FUNCTION_BLOCK FB_SlitPair_ISIS
VAR_INPUT
    nIdPositiveAxis: UINT; //ID of axis for which positive motion increases gap size
    nIdNegativeAxis: UINT; //ID of axis for which negative motion increases gap size
    nIdGapSizeAxis: UINT; //ID of virtual gap aperture size axis
    nIdGapCentreAxis: UINT; //ID of virtual gap centre position axis

    bEnable: BOOL; //Enable slit pair logic functionality
    bReset: BOOL; //Reset from error state
    fEncoderScaling: LREAL := 10000; //Virtual axis scaling denominator, default of 10000
    
    
    
END_VAR

//Linkable objects
VAR
    //Replacement limit links for real axes
    bPositiveAxis_FwdLimit AT %I* : BOOL;
    bPositiveAxis_BwdLimit AT %I* : BOOL;
    bNegativeAxis_FwdLimit AT %I* : BOOL;
    bNegativeAxis_BwdLimit AT %I* : BOOL;
    
    //Software encoders for virtual axes
    nGapSizeEncoder AT %Q*: UDINT := 0;
    nGapCentreEncoder AT %Q*: UDINT := 0;
END_VAR

VAR   
    fGapSize: LREAL;
    fGapCentre: LREAL;
    
    bAllHalted: BOOL := FALSE;
    bInternalResetHome: BOOL :=FALSE;

    fbSetpointGenEnablePositiveAxis: MC_ExtSetPointGenEnable;
    fbSetpointGenEnableNegativeAxis: MC_ExtSetPointGenEnable;
    fbSetpointGenEnableGapSizeAxis: MC_ExtSetPointGenEnable;
    fbSetpointGenEnableGapCentreAxis: MC_ExtSetPointGenEnable;

    fbSetpointGenDisablePositiveAxis: MC_ExtSetPointGenDisable;
    fbSetpointGenDisableNegativeAxis: MC_ExtSetPointGenDisable;
    fbSetpointGenDisableGapSizeAxis: MC_ExtSetPointGenDisable;
    fbSetpointGenDisableGapCentreAxis: MC_ExtSetPointGenDisable;

    fPosSetpointPositiveAxis: LREAL;
    fPosSetpointNegativeAxis: LREAL;
    fPosSetpointGapSizeAxis: LREAL;
    fPosSetpointGapCentreAxis: LREAL;
    
    fPosSetpointPositiveAxis_Nominal: LREAL;
    fPosSetpointNegativeAxis_Nominal: LREAL;
    fPosSetpointGapSizeAxis_Nominal: LREAL;
    fPosSetpointGapCentreAxis_Nominal: LREAL;

    fVeloSetpointPositiveAxis: LREAL;
    fVeloSetpointNegativeAxis: LREAL;
    fVeloSetpointGapSizeAxis: LREAL;
    fVeloSetpointGapCentreAxis: LREAL;

    fVeloSetpointPositiveAxis_Nominal: LREAL;
    fVeloSetpointNegativeAxis_Nominal: LREAL;
    fVeloSetpointGapSizeAxis_Nominal: LREAL;
    fVeloSetpointGapCentreAxis_Nominal: LREAL;
    
    nDirectionPositiveAxis: DINT;
    nDirectionNegativeAxis: DINT;
    nDirectionGapSizeAxis: DINT;
    nDirectionGapCentreAxis: DINT;
    
    ePositiveAxisState : E_AxisLimitState;
    eNegativeAxisState : E_AxisLimitState;
    eAxisPairState : E_SlitPairLimitState;
    

    eState: E_SlitPairStates := E_SlitPairStates.eInit;

    bInternalReset: BOOL;
    bHomingReset: BOOL := FALSE;

    //Two resets required due to homing functionality
    bResetInProgressCheck1: BOOL := FALSE;
    bResetInProgressCheck2: BOOL := FALSE;

    //internal MC_Reset, needed because the current reset in FB_Axis works only when there is an error. This should change once the reset functionality changes
    fbInternalResetTrig: R_TRIG;
    fbInternalResetHome: R_TRIG;
    fbResetPositiveAxis: MC_RESET;
    fbResetNegativeAxis: MC_RESET;
    fbResetGapSizeAxis: MC_RESET;
    fbResetGapCentreAxis: MC_RESET;
    fbResetHomedGap: MC_Home;
    fbResetHomedCentre: MC_Home;

END_VAR

(*SETUP INSTRUCTIONS
    All Axes:
        Allow motion commands to external setpoint axis := FALSE;
    Real Axes:
        Do not link limit switches to astAxes struct. Limits must be linked to FB_SlitPair_ISIS inputs
    Virtual axes:
        Encoder type set to Encoder (universal)
        Encoder mask set to 0xFFFFFFFF
        Encoder numerator/denominator scaling set to match FB fEncoderScaling value (default of 10 000 results in numerator of 0.0001 with denominator of 1)
        Link nDataIn1 of encoder to FB encoders
        Position lag monitoring can be left on
        Dynamics of virtual axes must be configured considering coupled mechanicals (e.g. don't set velocities your real axes can't achieve)
*)

//Limit switch passthrough by default - overridden where required in later logic to satisfy ExternalSetpointGenerators
GVL.astAxes[nIdPositiveAxis].stInputs.bLimitFwd:= bPositiveAxis_FwdLimit;
GVL.astAxes[nIdPositiveAxis].stInputs.bLimitBwd:= bPositiveAxis_BwdLimit;
GVL.astAxes[nIdNegativeAxis].stInputs.bLimitFwd:= bNegativeAxis_FwdLimit;
GVL.astAxes[nIdNegativeAxis].stInputs.bLimitBwd:= bNegativeAxis_BwdLimit;

//Enable Logic - Virtual axes automatically enable when real axes are enabled
actVirtualAxisEnable();

//Position of virtual axes
actVirtualAxisPositions();

//Determine limit state of real axes
actLimitState();

//Set fwEnabled and bwEnabled of virtual axes
actVirtualAxisLimits();

//Calculate position and velocity setpoints
actCalculateSetpointPositionAndVelocity();

//Calculate direction setpoints
actCalculateSetpointDirections();




//Error state handling - only handle errors that disable motion
IF bEnable AND (GVL.astAxes[nIdPositiveAxis].Axis.Status.ErrorStop OR GVL.astAxes[nIdNegativeAxis].Axis.Status.ErrorStop OR GVL.astAxes[nIdGapSizeAxis].Axis.Status.ErrorStop OR GVL.astAxes[nIdGapCentreAxis].Axis.Status.ErrorStop) THEN
    eState := E_SlitPairStates.eError;
END_IF

//Propagate real axis error to virtual
IF GVL.astAxes[nIdPositiveAxis].Axis.Status.ErrorStop AND (NOT GVL.astAxes[nIdGapSizeAxis].Axis.Status.ErrorStop OR NOT GVL.astAxes[nIdGapCentreAxis].Axis.Status.ErrorStop) THEN
    GVL.astAxes[nIdGapSizeAxis].stStatus.bError := TRUE;
    GVL.astAxes[nIdGapCentreAxis].stStatus.bError := TRUE;
    GVL.astAxes[nIdGapSizeAxis].stStatus.nErrorID := GVL.astAxes[nIdPositiveAxis].stStatus.nErrorID;
    GVL.astAxes[nIdGapCentreAxis].stStatus.nErrorID := GVL.astAxes[nIdPositiveAxis].stStatus.nErrorID;
ELSIF  GVL.astAxes[nIdNegativeAxis].Axis.Status.ErrorStop AND (NOT GVL.astAxes[nIdGapSizeAxis].Axis.Status.ErrorStop OR NOT GVL.astAxes[nIdGapCentreAxis].Axis.Status.ErrorStop) THEN
    GVL.astAxes[nIdGapSizeAxis].stStatus.bError := TRUE;
    GVL.astAxes[nIdGapCentreAxis].stStatus.bError := TRUE;
    GVL.astAxes[nIdGapSizeAxis].stStatus.nErrorID := GVL.astAxes[nIdNegativeAxis].stStatus.nErrorID;
    GVL.astAxes[nIdGapCentreAxis].stStatus.nErrorID := GVL.astAxes[nIdNegativeAxis].stStatus.nErrorID;
END_IF

//Internal Reset linked to any axis reset
bInternalReset := bReset OR GVL.astAxes[nIdPositiveAxis].stControl.bReset OR GVL.astAxes[nIdNegativeAxis].stControl.bReset OR GVL.astAxes[nIdGapSizeAxis].stControl.bReset OR GVL.astAxes[nIdGapCentreAxis].stControl.bReset;

//If real axis is homing, change state
IF bEnable AND (GVL.astAxes[nIdPositiveAxis].Axis.Status.HomingBusy OR GVL.astAxes[nIdNegativeAxis].Axis.Status.HomingBusy) THEN
    eState := E_SlitPairStates.eWaitForRealHomed;
END_IF

//Link all halt buttons in motors
IF GVL.astAxes[nIdPositiveAxis].stControl.bHalt OR GVL.astAxes[nIdNegativeAxis].stControl.bHalt OR
    GVL.astAxes[nIdGapSizeAxis].stControl.bHalt OR GVL.astAxes[nIdGapCentreAxis].stControl.bHalt THEN
    actHaltAllAxes();   //Will upset setpoint generator axes - may be able to fix by only issuing to non-setpoint generated axes
END_IF

//Propagate homing status
fbResetHomedGap(Axis:= GVL.astAxes[nIdGapSizeAxis].Axis, HomingMode:= MC_ResetCalibration);
fbResetHomedCentre(Axis:= GVL.astAxes[nIdGapCentreAxis].Axis, HomingMode:= MC_ResetCalibration);
fbInternalResetHome(CLK:= fbResetHomedCentre.Done OR fbResetHomedGap.Done );

IF NOT GVL.astAxes[nIdPositiveAxis].stStatus.bHomed OR NOT GVL.astAxes[nIdNegativeAxis].stStatus.bHomed THEN
        fbResetHomedGap.Execute := TRUE;
        fbResetHomedCentre.Execute := TRUE;
END_IF

IF fbInternalResetHome.Q THEN
        fbResetHomedGap.Execute := FALSE;
        fbResetHomedCentre.Execute := FALSE;
END_IF


//State machine
IF bEnable THEN
    CASE eState OF  //HOMING LOOP ISSUE
        E_SlitPairStates.eInit:
            //If real axes are calibrated, then home the virtual axes, else go Operatioanl
            fbResetPositiveAxis(Axis:=GVL.astAxes[nIdPositiveAxis].Axis, Execute:=FALSE);
            fbResetNegativeAxis(Axis:=GVL.astAxes[nIdNegativeAxis].Axis, Execute:=FALSE);
            fbResetGapSizeAxis(Axis:=GVL.astAxes[nIdGapSizeAxis].Axis, Execute:=FALSE);
            fbResetGapCentreAxis(Axis:=GVL.astAxes[nIdGapCentreAxis].Axis, Execute:=FALSE);
            IF GVL.astAxes[nIdPositiveAxis].stStatus.bHomed AND GVL.astAxes[nIdNegativeAxis].stStatus.bHomed THEN
               GVL.astAxes[nIdGapSizeAxis].stConfig.eHomeSeq := E_HomingRoutines.eHomeDirect;
               GVL.astAxes[nIdGapCentreAxis].stConfig.eHomeSeq := E_HomingRoutines.eHomeDirect;
               GVL.astAxes[nIdGapSizeAxis].stConfig.fHomePosition := fGapSize;
               GVL.astAxes[nIdGapCentreAxis].stConfig.fHomePosition := fGapCentre;
                eState := E_SlitPairStates.eWaitForVirtualHomed;
            ELSE
                eState := E_SlitPairStates.eOperational;
            END_IF

        E_SlitPairStates.eWaitForVirtualHomed:
            //Wait for virtual axis homing to complete/
            GVL.astAxes[nIdGapSizeAxis].stControl.eCommand := E_MotionFunctions.eHome;
            GVL.astAxes[nIdGapSizeAxis].stControl.bExecute := TRUE;
            GVL.astAxes[nIdGapCentreAxis].stControl.eCommand := E_MotionFunctions.eHome;
            GVL.astAxes[nIdGapCentreAxis].stControl.bExecute := TRUE;
            IF GVL.astAxes[nIdGapSizeAxis].stStatus.bHomed AND GVL.astAxes[nIdGapCentreAxis].stStatus.bHomed THEN
                eState := E_SlitPairStates.eOperational;
            END_IF
            //IF NOT IN HOMING STATE

        E_SlitPairStates.eOperational:
            bResetInProgressCheck1 := FALSE;
            //Detect whether real or virtual axes are moving
            IF GVL.astAxes[nIdGapSizeAxis].stStatus.bMoving OR GVL.astAxes[nIdGapCentreAxis].stStatus.bMoving THEN
                eState := E_SlitPairStates.eEnableRealGenerators;
            END_IF
            IF GVL.astAxes[nIdPositiveAxis].stStatus.bMoving OR GVL.astAxes[nIdNegativeAxis].stStatus.bMoving THEN
                eState := E_SlitPairStates.eEnableVirtualGenerators;
            END_IF

        E_SlitPairStates.eEnableRealGenerators:
            //Temporary override of limits
            GVL.astAxes[nIdPositiveAxis].stInputs.bLimitFwd:= TRUE;
            GVL.astAxes[nIdPositiveAxis].stInputs.bLimitBwd:= TRUE;
            GVL.astAxes[nIdNegativeAxis].stInputs.bLimitFwd:= TRUE;
            GVL.astAxes[nIdNegativeAxis].stInputs.bLimitBwd:= TRUE;
            fbSetpointGenEnablePositiveAxis.Execute := TRUE;
            fbSetpointGenEnableNegativeAxis.Execute := TRUE;
            eState := E_SlitPairStates.eCheckRealAxisGeneratorsEnabled;

        E_SlitPairStates.eCheckRealAxisGeneratorsEnabled:
            //Hold MC_Power on until generators have enabled           
            IF fbSetpointGenEnablePositiveAxis.Enabled AND fbSetpointGenEnableNegativeAxis.Enabled THEN
                eState := E_SlitPairStates.eWaitForVirtualMoveDone;
            END_IF

        E_SlitPairStates.eWaitForVirtualMoveDone:            
            IF NOT(GVL.astAxes[nIdGapSizeAxis].stStatus.bMoving OR GVL.astAxes[nIdGapCentreAxis].stStatus.bMoving) THEN
                eState := E_SlitPairStates.eDisableRealGenerators;
            END_IF

        E_SlitPairStates.eDisableRealGenerators:
            fbSetpointGenDisablePositiveAxis.Execute := TRUE;
            fbSetpointGenDisableNegativeAxis.Execute := TRUE;
            eState := E_SlitPairStates.eOperational;

        E_SlitPairStates.eEnableVirtualGenerators:
            //Hold MC_Power on until generators have enabled
            GVL.astAxes[nIdPositiveAxis].stInputs.bLimitFwd:= TRUE;
            GVL.astAxes[nIdPositiveAxis].stInputs.bLimitBwd:= TRUE;
            GVL.astAxes[nIdNegativeAxis].stInputs.bLimitFwd:= TRUE;
            GVL.astAxes[nIdNegativeAxis].stInputs.bLimitBwd:= TRUE;
            fbSetpointGenEnableGapSizeAxis.Execute := TRUE;
            fbSetpointGenEnableGapCentreAxis.Execute := TRUE;
            eState := E_SlitPairStates.eCheckVirtualAxisGeneratorsEnabled;

        E_SlitPairStates.eCheckVirtualAxisGeneratorsEnabled:
            //Hold MC_Power on until generators have enabled
            IF fbSetpointGenEnableGapSizeAxis.Enabled AND fbSetpointGenEnableGapCentreAxis.Enabled THEN
                eState := E_SlitPairStates.eWaitForRealMoveDone;
            END_IF

        E_SlitPairStates.eWaitForRealMoveDone:
            IF NOT(GVL.astAxes[nIdPositiveAxis].stStatus.bMoving OR GVL.astAxes[nIdNegativeAxis].stStatus.bMoving) THEN
                eState := E_SlitPairStates.eDisableVirtualGenerators;
            END_IF

        E_SlitPairStates.eDisableVirtualGenerators:
            fbSetpointGenDisableGapSizeAxis.Execute := TRUE;
            fbSetpointGenDisableGapCentreAxis.Execute := TRUE;
            eState := E_SlitPairStates.eOperational;

        E_SlitPairStates.eError:
            actHaltAllAxes();

            IF bHomingReset THEN
                bInternalReset := TRUE;
                bResetInProgressCheck1 := TRUE;
                bResetInProgressCheck2 := TRUE;
                bHomingReset := FALSE;
            END_IF
            IF bInternalReset OR bReset OR bResetInProgressCheck2 THEN
                fbResetPositiveAxis(Axis:=GVL.astAxes[nIdPositiveAxis].Axis, Execute:=TRUE);
                fbResetNegativeAxis(Axis:=GVL.astAxes[nIdNegativeAxis].Axis, Execute:=TRUE);
                fbResetGapSizeAxis(Axis:=GVL.astAxes[nIdGapSizeAxis].Axis, Execute:=TRUE);
                fbResetGapCentreAxis(Axis:=GVL.astAxes[nIdGapCentreAxis].Axis, Execute:=TRUE);
                GVL.astAxes[nIdPositiveAxis].stControl.bReset := TRUE;
                GVL.astAxes[nIdNegativeAxis].stControl.bReset := TRUE;
                GVL.astAxes[nIdGapSizeAxis].stControl.bReset := TRUE;
                GVL.astAxes[nIdGapCentreAxis].stControl.bReset := TRUE;
                IF NOT(bResetInProgressCheck1) THEN
                    bResetInProgressCheck2 := FALSE;
                END_IF
            END_IF

            IF NOT(GVL.astAxes[nIdPositiveAxis].stStatus.bError) AND NOT(GVL.astAxes[nIdNegativeAxis].stStatus.bError) AND NOT(GVL.astAxes[nIdGapSizeAxis].stStatus.bError) AND NOT(GVL.astAxes[nIdGapCentreAxis].stStatus.bError) THEN
                eState := E_SlitPairStates.eInit;
            END_IF

        E_SlitPairStates.eWaitForRealHomed:
            bHomingReset := TRUE;
            IF NOT GVL.astAxes[nIdPositiveAxis].Axis.Status.Homed OR NOT GVL.astAxes[nIdNegativeAxis].Axis.Status.Homed THEN
                eState := E_SlitPairStates.eInit;
            END_IF
    END_CASE
END_IF

//Call spGenerator FBs
actGeneratorEnableDisable();

//Feed externalsetpoint generators setpoint values - ignoring acceleration
MC_ExtSetPointGenFeed(Axis:= GVL.astAxes[nIdPositiveAxis].Axis, Position:= fPosSetpointPositiveAxis, Velocity:= fVeloSetpointPositiveAxis, Acceleration:= 0, Direction:= nDirectionPositiveAxis);
MC_ExtSetPointGenFeed(Axis:= GVL.astAxes[nIdNegativeAxis].Axis, Position:= fPosSetpointNegativeAxis, Velocity:= fVeloSetpointNegativeAxis, Acceleration:= 0, Direction:= nDirectionNegativeAxis);
MC_ExtSetPointGenFeed(Axis:= GVL.astAxes[nIdGapSizeAxis].Axis, Position:= fPosSetpointGapSizeAxis, Velocity:= fVeloSetpointGapSizeAxis, Acceleration:= 0, Direction:= nDirectionGapSizeAxis);
MC_ExtSetPointGenFeed(Axis:= GVL.astAxes[nIdGapCentreAxis].Axis, Position:= fPosSetpointGapCentreAxis, Velocity:= fVeloSetpointGapCentreAxis, Acceleration:= 0, Direction:= nDirectionGapCentreAxis);

bReset := FALSE;

ACTION actCalculateSetpointDirections:
IF fVeloSetpointPositiveAxis > 0 THEN
    nDirectionPositiveAxis := 1; //moving forward
ELSIF fVeloSetpointPositiveAxis < 0 THEN
    nDirectionPositiveAxis := -1; //moving backward
ELSE
    nDirectionPositiveAxis := 0; //stationary
END_IF

IF fVeloSetpointNegativeAxis > 0 THEN
    nDirectionNegativeAxis := 1; //moving forward
ELSIF fVeloSetpointNegativeAxis < 0 THEN
    nDirectionNegativeAxis := -1; //moving backward
ELSE
    nDirectionNegativeAxis := 0; //stationary
END_IF

IF fVeloSetpointGapSizeAxis > 0 THEN
    nDirectionGapSizeAxis := 1; //moving forward
ELSIF fVeloSetpointGapSizeAxis < 0 THEN
    nDirectionGapSizeAxis := -1; //moving backward
ELSE
    nDirectionGapSizeAxis := 0; //stationary
END_IF

IF fVeloSetpointGapCentreAxis > 0 THEN
    nDirectionGapCentreAxis := 1; //moving forward
ELSIF fVeloSetpointGapCentreAxis < 0 THEN
    nDirectionGapCentreAxis := -1; //moving backward
ELSE
    nDirectionGapCentreAxis := 0; //stationary
END_IF
END_ACTION

ACTION actCalculateSetpointPositionAndVelocity:
//Axis status update to get current NC move progress
GVL.astAxes[nIdPositiveAxis].Axis.ReadStatus();
GVL.astAxes[nIdNegativeAxis].Axis.ReadStatus();
GVL.astAxes[nIdGapSizeAxis].Axis.ReadStatus();
GVL.astAxes[nIdGapCentreAxis].Axis.ReadStatus();


//Calculate nominal setpoint positions assuming no limits
fPosSetpointPositiveAxis_Nominal := GVL.astAxes[nIdGapCentreAxis].Axis.NcToPlc.SetPos + (GVL.astAxes[nIdGapSizeAxis].Axis.NcToPlc.SetPos/2);
fPosSetpointNegativeAxis_Nominal := GVL.astAxes[nIdGapCentreAxis].Axis.NcToPlc.SetPos - (GVL.astAxes[nIdGapSizeAxis].Axis.NcToPlc.SetPos/2);
fPosSetpointGapSizeAxis_Nominal := GVL.astAxes[nIdPositiveAxis].Axis.NcToPlc.SetPos - GVL.astAxes[nIdNegativeAxis].Axis.NcToPlc.SetPos;
fPosSetpointGapCentreAxis_Nominal := (GVL.astAxes[nIdPositiveAxis].Axis.NcToPlc.SetPos + GVL.astAxes[nIdNegativeAxis].Axis.NcToPlc.SetPos) / 2;

//Calculate nominal setpoint velocities assuming no limits
fVeloSetpointPositiveAxis_Nominal := GVL.astAxes[nIdGapCentreAxis].Axis.NcToPlc.SetVelo +(GVL.astAxes[nIdGapSizeAxis].Axis.NcToPlc.SetVelo/2);
fVeloSetpointNegativeAxis_Nominal := GVL.astAxes[nIdGapCentreAxis].Axis.NcToPlc.SetVelo -(GVL.astAxes[nIdGapSizeAxis].Axis.NcToPlc.SetVelo/2);
fVeloSetpointGapSizeAxis_Nominal := GVL.astAxes[nIdPositiveAxis].Axis.NcToPlc.SetVelo - GVL.astAxes[nIdNegativeAxis].Axis.NcToPlc.SetVelo;
fVeloSetpointGapCentreAxis_Nominal := GVL.astAxes[nIdPositiveAxis].Axis.NcToPlc.SetVelo + GVL.astAxes[nIdNegativeAxis].Axis.NcToPlc.SetVelo;


//Detect IF moving in Virtual axis gap control mode
IF GVL.astAxes[nIdPositiveAxis].Axis.Status.ExtSetPointGenEnabled OR GVL.astAxes[nIdNegativeAxis].Axis.Status.ExtSetPointGenEnabled THEN
    //IF gap size getting bigger
    IF GVL.astAxes[nIdGapSizeAxis].Axis.Status.PositiveDirection THEN
        CASE eAxisPairState OF            
        E_SlitPairLimitState.PositiveOnForward_NegativeOnForward:   Setpoint_PositiveDisabled();            
        E_SlitPairLimitState.PositiveOnForward_NegativeOnBackward:  Setpoint_AllDisabled();            
        E_SlitPairLimitState.PositiveOnForward_NegativeOnNoLimit:   Setpoint_PositiveDisabled();            
        E_SlitPairLimitState.PositiveOnBackward_NegativeOnForward:  Setpoint_Normal();            
        E_SlitPairLimitState.PositiveOnBackward_NegativeOnBackward: Setpoint_NegativeDisabled();            
        E_SlitPairLimitState.PositiveOnBackward_NegativeOnNoLimit:  Setpoint_Normal();            
        E_SlitPairLimitState.PositiveOnNoLimit_NegativeOnForward:   Setpoint_Normal();            
        E_SlitPairLimitState.PositiveOnNoLimit_NegativeOnBackward:  Setpoint_NegativeDisabled();            
        E_SlitPairLimitState.PositiveOnNoLimit_NegativeOnNoLimit:   Setpoint_Normal();
        END_CASE
    //IF gap size getting smaller
    ELSIF GVL.astAxes[nIdGapSizeAxis].Axis.Status.NegativeDirection THEN
        CASE eAxisPairState OF            
        E_SlitPairLimitState.PositiveOnForward_NegativeOnForward:   Setpoint_NegativeDisabled();
        E_SlitPairLimitState.PositiveOnForward_NegativeOnBackward:  Setpoint_Normal();
        E_SlitPairLimitState.PositiveOnForward_NegativeOnNoLimit:   Setpoint_Normal();
        E_SlitPairLimitState.PositiveOnBackward_NegativeOnForward:  Setpoint_AllDisabled();            
        E_SlitPairLimitState.PositiveOnBackward_NegativeOnBackward: Setpoint_PositiveDisabled();            
        E_SlitPairLimitState.PositiveOnBackward_NegativeOnNoLimit:  Setpoint_PositiveDisabled();
        E_SlitPairLimitState.PositiveOnNoLimit_NegativeOnForward:   Setpoint_NegativeDisabled();           
        E_SlitPairLimitState.PositiveOnNoLimit_NegativeOnBackward:  Setpoint_Normal();
        E_SlitPairLimitState.PositiveOnNoLimit_NegativeOnNoLimit:   Setpoint_Normal();                       
        END_CASE
    ELSE //Gap size axis is stationary
        //IF gap centre moving in positive direction
        IF GVL.astAxes[nIdGapCentreAxis].Axis.Status.PositiveDirection THEN
            CASE eAxisPairState OF            
            E_SlitPairLimitState.PositiveOnForward_NegativeOnForward:   Setpoint_AllDisabled();
            E_SlitPairLimitState.PositiveOnForward_NegativeOnBackward:  Setpoint_AllDisabled();           
            E_SlitPairLimitState.PositiveOnForward_NegativeOnNoLimit:   Setpoint_AllDisabled();            
            E_SlitPairLimitState.PositiveOnBackward_NegativeOnForward:  Setpoint_AllDisabled();           
            E_SlitPairLimitState.PositiveOnBackward_NegativeOnBackward: Setpoint_Normal();            
            E_SlitPairLimitState.PositiveOnBackward_NegativeOnNoLimit:  Setpoint_Normal();            
            E_SlitPairLimitState.PositiveOnNoLimit_NegativeOnForward:   Setpoint_AllDisabled();            
            E_SlitPairLimitState.PositiveOnNoLimit_NegativeOnBackward:  Setpoint_Normal();            
            E_SlitPairLimitState.PositiveOnNoLimit_NegativeOnNoLimit:   Setpoint_Normal();                       
            END_CASE
        //IF gap centre moving in negative direction
        ELSIF GVL.astAxes[nIdGapCentreAxis].Axis.Status.NegativeDirection THEN
            CASE eAxisPairState OF            
            E_SlitPairLimitState.PositiveOnForward_NegativeOnForward:   Setpoint_Normal();
            E_SlitPairLimitState.PositiveOnForward_NegativeOnBackward:  Setpoint_AllDisabled();            
            E_SlitPairLimitState.PositiveOnForward_NegativeOnNoLimit:   Setpoint_Normal();            
            E_SlitPairLimitState.PositiveOnBackward_NegativeOnForward:  Setpoint_AllDisabled();            
            E_SlitPairLimitState.PositiveOnBackward_NegativeOnBackward: Setpoint_AllDisabled();            
            E_SlitPairLimitState.PositiveOnBackward_NegativeOnNoLimit:  Setpoint_AllDisabled();            
            E_SlitPairLimitState.PositiveOnNoLimit_NegativeOnForward:   Setpoint_Normal();            
            E_SlitPairLimitState.PositiveOnNoLimit_NegativeOnBackward:  Setpoint_AllDisabled();            
            E_SlitPairLimitState.PositiveOnNoLimit_NegativeOnNoLimit:   Setpoint_Normal();                       
            END_CASE
		END_IF
    END_IF
END_IF

//Detect IF real axis control. Normal operation as no limits on virtual axes
IF GVL.astAxes[nIdGapCentreAxis].Axis.Status.ExtSetPointGenEnabled AND GVL.astAxes[nIdGapSizeAxis].Axis.Status.ExtSetPointGenEnabled THEN
    fPosSetpointGapSizeAxis := GVL.astAxes[nIdPositiveAxis].Axis.NcToPlc.SetPos - GVL.astAxes[nIdNegativeAxis].Axis.NcToPlc.SetPos;
    fPosSetpointGapCentreAxis := (GVL.astAxes[nIdPositiveAxis].Axis.NcToPlc.SetPos + GVL.astAxes[nIdNegativeAxis].Axis.NcToPlc.SetPos) / 2;
    fVeloSetpointGapCentreAxis := fVeloSetpointGapCentreAxis_Nominal;
    fVeloSetpointGapSizeAxis := fVeloSetpointGapSizeAxis_Nominal;
END_IF
END_ACTION

ACTION actGeneratorEnableDisable:

fbSetpointGenEnablePositiveAxis(Axis:=GVL.astAxes[nIdPositiveAxis].Axis);
fbSetpointGenEnablePositiveAxis.Execute := FALSE;

fbSetpointGenEnableNegativeAxis(Axis:=GVL.astAxes[nIdNegativeAxis].Axis);
fbSetpointGenEnableNegativeAxis.Execute := FALSE;

fbSetpointGenEnableGapSizeAxis(Axis:=GVL.astAxes[nIdGapSizeAxis].Axis);
fbSetpointGenEnableGapSizeAxis.Execute := FALSE;

fbSetpointGenEnableGapCentreAxis(Axis:=GVL.astAxes[nIdGapCentreAxis].Axis);
fbSetpointGenEnableGapCentreAxis.Execute := FALSE;


fbSetpointGenDisablePositiveAxis(Axis:=GVL.astAxes[nIdPositiveAxis].Axis);
fbSetpointGenDisablePositiveAxis.Execute := FALSE;

fbSetpointGenDisableNegativeAxis(Axis:=GVL.astAxes[nIdNegativeAxis].Axis);
fbSetpointGenDisableNegativeAxis.Execute := FALSE;

fbSetpointGenDisableGapSizeAxis(Axis:=GVL.astAxes[nIdGapSizeAxis].Axis);
fbSetpointGenDisableGapSizeAxis.Execute := FALSE;

fbSetpointGenDisableGapCentreAxis(Axis:=GVL.astAxes[nIdGapCentreAxis].Axis);
fbSetpointGenDisableGapCentreAxis.Execute := FALSE;
END_ACTION

ACTION actHaltAllAxes:
GVL.astAxes[nIdPositiveAxis].stControl.bHalt := TRUE;
GVL.astAxes[nIdNegativeAxis].stControl.bHalt := TRUE;
GVL.astAxes[nIdGapSizeAxis].stControl.bHalt := TRUE;
GVL.astAxes[nIdGapCentreAxis].stControl.bHalt := TRUE;
bAllHalted := TRUE;

//Reset Halts
IF bAllHalted AND NOT GVL.astAxes[nIdPositiveAxis].stStatus.bMoving AND NOT GVL.astAxes[nIdNegativeAxis].stStatus.bMoving
 AND NOT GVL.astAxes[nIdGapSizeAxis].stStatus.bMoving AND NOT GVL.astAxes[nIdGapCentreAxis].stStatus.bMoving THEN
   GVL.astAxes[nIdPositiveAxis].stControl.bHalt := FALSE;
   GVL.astAxes[nIdNegativeAxis].stControl.bHalt := FALSE;
   GVL.astAxes[nIdGapSizeAxis].stControl.bHalt := FALSE;
   GVL.astAxes[nIdGapCentreAxis].stControl.bHalt := FALSE;
   bAllHalted := FALSE;
END_IF
END_ACTION

ACTION actLimitState:
//Positive axis state
IF bPositiveAxis_FwdLimit = FALSE THEN
    ePositiveAxisState := E_AxisLimitState.OnForwardLimit;
ELSIF bPositiveAxis_BwdLimit = FALSE THEN
    ePositiveAxisState := E_AxisLimitState.OnBackwardLimit;
ELSE
    ePositiveAxisState := E_AxisLimitState.NoLimit;
END_IF

//Negative axis state
IF bNegativeAxis_FwdLimit = FALSE THEN
    eNegativeAxisState := E_AxisLimitState.OnForwardLimit;
ELSIF bNegativeAxis_BwdLimit = FALSE THEN
    eNegativeAxisState := E_AxisLimitState.OnBackwardLimit;
ELSE
    eNegativeAxisState := E_AxisLimitState.NoLimit;
END_IF

//Combined slit pair limit state
CASE ePositiveAxisState OF
    E_AxisLimitState.OnForwardLimit:
        CASE eNegativeAxisState OF
            E_AxisLimitState.OnForwardLimit:
                eAxisPairState := E_SlitPairLimitState.PositiveOnForward_NegativeOnForward;
            E_AxisLimitState.OnBackwardLimit:
                eAxisPairState := E_SlitPairLimitState.PositiveOnForward_NegativeOnBackward;
            E_AxisLimitState.NoLimit:
                eAxisPairState := E_SlitPairLimitState.PositiveOnForward_NegativeOnNoLimit;            
		END_CASE
    E_AxisLimitState.OnBackwardLimit:
        CASE eNegativeAxisState OF
            E_AxisLimitState.OnForwardLimit:
                eAxisPairState := E_SlitPairLimitState.PositiveOnBackward_NegativeOnForward;
            E_AxisLimitState.OnBackwardLimit:
                eAxisPairState := E_SlitPairLimitState.PositiveOnBackward_NegativeOnBackward;
            E_AxisLimitState.NoLimit:
                eAxisPairState := E_SlitPairLimitState.PositiveOnBackward_NegativeOnNoLimit;            
		END_CASE
    E_AxisLimitState.NoLimit:
        CASE eNegativeAxisState OF
            E_AxisLimitState.OnForwardLimit:
                eAxisPairState := E_SlitPairLimitState.PositiveOnNoLimit_NegativeOnForward;
            E_AxisLimitState.OnBackwardLimit:
                eAxisPairState := E_SlitPairLimitState.PositiveOnNoLimit_NegativeOnBackward;
            E_AxisLimitState.NoLimit:
                eAxisPairState := E_SlitPairLimitState.PositiveOnNoLimit_NegativeOnNoLimit;            
		END_CASE
END_CASE
END_ACTION

ACTION actVirtualAxisEnable:
GVL.astAxes[nIdGapSizeAxis].stControl.bEnable := GVL.astAxes[nIdPositiveAxis].stControl.bEnable AND GVL.astAxes[nIdNegativeAxis].stControl.bEnable;
GVL.astAxes[nIdGapCentreAxis].stControl.bEnable := GVL.astAxes[nIdPositiveAxis].stControl.bEnable AND GVL.astAxes[nIdNegativeAxis].stControl.bEnable;
END_ACTION

ACTION actVirtualAxisLimits:
//Gap size forward limit
IF GVL.astAxes[nIdPositiveAxis].stStatus.bFwEnabled = FALSE AND GVL.astAxes[nIdNegativeAxis].stStatus.bBwEnabled = FALSE THEN
    GVL.astAxes[nIdGapSizeAxis].stStatus.bFwEnabled := FALSE;
ELSE
    GVL.astAxes[nIdGapSizeAxis].stStatus.bFwEnabled := TRUE;
END_IF

//Gap size backward limit
IF GVL.astAxes[nIdPositiveAxis].stStatus.bBwEnabled = FALSE AND GVL.astAxes[nIdNegativeAxis].stStatus.bFwEnabled = FALSE THEN
    GVL.astAxes[nIdGapSizeAxis].stStatus.bBwEnabled := FALSE;
ELSE
    GVL.astAxes[nIdGapSizeAxis].stStatus.bBwEnabled := TRUE;
END_IF

//Gap centre forward limit
IF GVL.astAxes[nIdPositiveAxis].stStatus.bFwEnabled = FALSE OR GVL.astAxes[nIdNegativeAxis].stStatus.bFwEnabled = FALSE THEN
    GVL.astAxes[nIdGapCentreAxis].stStatus.bFwEnabled := FALSE;
ELSE
    GVL.astAxes[nIdGapCentreAxis].stStatus.bFwEnabled := TRUE;
END_IF

//Gap centre backward limit
IF GVL.astAxes[nIdPositiveAxis].stStatus.bBwEnabled = FALSE OR GVL.astAxes[nIdNegativeAxis].stStatus.bBwEnabled = FALSE THEN
    GVL.astAxes[nIdGapCentreAxis].stStatus.bBwEnabled := FALSE;
ELSE
    GVL.astAxes[nIdGapCentreAxis].stStatus.bBwEnabled := TRUE;
END_IF
END_ACTION

ACTION actVirtualAxisPositions:
(*Calculate virtual axis positions and convert to UDINT.
Conversion to UDINT is prohibited if it would exceed UDINT max value of 4,294,967,295.
If this is not done, it can cause overflow when connected to the encoder input and hard-crash the PLC which will only recover with a power cycle.
To preserve decimal position data of the LREAL (i.e. anything <1mm) it is necessary to scale the value before converting to UDINT.
This can be reversed with the correct scaling at the NC encoder level.
*)
fGapSize := GVL.astAxes[nIdPositiveAxis].stStatus.fActPosition - GVL.astAxes[nIdNegativeAxis].stStatus.fActPosition;
fGapCentre := (GVL.astAxes[nIdPositiveAxis].stStatus.fActPosition + GVL.astAxes[nIdNegativeAxis].stStatus.fActPosition)/2;

IF ABS(fGapSize) < 100000 THEN
    nGapSizeEncoder := LREAL_TO_UDINT(fGapSize*fEncoderScaling);
END_IF
IF ABS(fGapCentre) < 100000 THEN
    nGapCentreEncoder := LREAL_TO_UDINT(fGapCentre*fEncoderScaling);
END_IF
END_ACTION

ACTION Setpoint_AllDisabled:
fPosSetpointPositiveAxis := fPosSetpointPositiveAxis;
fPosSetpointNegativeAxis := fPosSetpointNegativeAxis;            
fVeloSetpointPositiveAxis := 0;
fVeloSetpointNegativeAxis := 0;

fbSetpointGenEnableGapCentreAxis.Execute:= TRUE;
fbSetpointGenEnableGapCentreAxis(Axis:= GVL.astAxes[nIdGapCentreAxis].Axis);
fPosSetpointGapCentreAxis := (GVL.astAxes[nIdPositiveAxis].Axis.NcToPlc.ActPos + GVL.astAxes[nIdNegativeAxis].Axis.NcToPlc.ActPos)/2;
fVeloSetpointGapCentreAxis := fVeloSetpointGapCentreAxis_Nominal;

actHaltAllAxes();
END_ACTION

ACTION Setpoint_NegativeDisabled:
fPosSetpointPositiveAxis := GVL.astAxes[nIdGapSizeAxis].Axis.NcToPlc.SetPos + GVL.astAxes[nIdNegativeAxis].Axis.NcToPlc.ActPos;
fPosSetpointNegativeAxis := fPosSetpointNegativeAxis;
fVeloSetpointPositiveAxis := GVL.astAxes[nIdGapSizeAxis].Axis.NcToPlc.SetVelo;
fVeloSetpointNegativeAxis := 0;
            
fbSetpointGenEnableGapCentreAxis.Execute:= TRUE;
fbSetpointGenEnableGapCentreAxis(Axis:= GVL.astAxes[nIdGapCentreAxis].Axis);
fPosSetpointGapCentreAxis := fGapCentre;
fVeloSetpointGapCentreAxis := fVeloSetpointGapCentreAxis_Nominal;

GVL.astAxes[nIdGapSizeAxis].stConfig.fOverride:=50;
END_ACTION

ACTION Setpoint_Normal:
fPosSetpointPositiveAxis := fPosSetpointPositiveAxis_Nominal;
fPosSetpointNegativeAxis := fPosSetpointNegativeAxis_Nominal;
fVeloSetpointPositiveAxis := fVeloSetpointPositiveAxis_Nominal;
fVeloSetpointNegativeAxis := fVeloSetpointNegativeAxis_Nominal;

GVL.astAxes[nIdGapSizeAxis].stConfig.fOverride:=100;
END_ACTION

ACTION Setpoint_PositiveDisabled:
fPosSetpointPositiveAxis := fPosSetpointPositiveAxis;
fPosSetpointNegativeAxis := GVL.astAxes[nIdPositiveAxis].Axis.NcToPlc.ActPos - GVL.astAxes[nIdGapSizeAxis].Axis.NcToPlc.SetPos;
fVeloSetpointPositiveAxis := 0;
fVeloSetpointNegativeAxis := GVL.astAxes[nIdGapSizeAxis].Axis.NcToPlc.SetVelo;
            
fbSetpointGenEnableGapCentreAxis.Execute:= TRUE;
fbSetpointGenEnableGapCentreAxis(Axis:= GVL.astAxes[nIdGapCentreAxis].Axis);
fPosSetpointGapCentreAxis := fGapCentre;
fVeloSetpointGapCentreAxis := fVeloSetpointGapCentreAxis_Nominal;

GVL.astAxes[nIdGapSizeAxis].stConfig.fOverride:=50;
END_ACTION

END_FUNCTION_BLOCK

(* stored: Version 1.1.0.1, ProductVersion 3.1.4024.11
   POU FB_SlitPair_ISIS: Id {b3c09412-d9b8-4fdb-95f8-f2ca5d9e6945}, SpecialFunc None
   Folder Setpoint_Generator_Actions: Id {8e494922-e7c2-4daa-80b3-ea89aa78df74}
   Action actCalculateSetpointDirections: Id {5abf4283-d432-4b19-be96-a15b54858b40}
   Action actCalculateSetpointPositionAndVelocity: Id {1756795d-6a25-4bcd-9ca1-dcd9ccd9b4a7}
   Action actGeneratorEnableDisable: Id {3488c74c-bc18-48be-a44b-85fc45e9d726}
   Action actHaltAllAxes: Id {b7970e1d-c1fa-487e-a0a7-5d7f0550df46}
   Action actLimitState: Id {0bf1ea49-b548-4e60-a8eb-6a1e52eb2a32}
   Action actVirtualAxisEnable: Id {9800ad84-33b1-45e1-8f1c-18ce4e663f2f}
   Action actVirtualAxisLimits: Id {b46f168f-6065-4588-af1f-8e4bf3d9b991}
   Action actVirtualAxisPositions: Id {728f3665-a1f5-47e1-9096-f32eff42a946}
   Action Setpoint_AllDisabled: Id {8d0131b7-d925-4748-8e58-1076d969b851}
   Action Setpoint_NegativeDisabled: Id {9ce73458-d767-47d6-a68a-e8346e22f1ca}
   Action Setpoint_Normal: Id {2ee67b84-83cd-44fc-84d0-218d8dc38cfa}
   Action Setpoint_PositiveDisabled: Id {1b4e9e96-8a89-4887-bc05-9c26a4b38f02} *)
